PROGRAM MAIN
VAR
	fbEvent:				FB_Event;
	fbEventHandler:			FB_EventHandler;
	fbTcLoggerHandler:		FB_TcLoggerHandler;	
	fbEmergencyHandler:		FB_EmergencyHandler;
	bInit:					BOOL:= TRUE;
	bDebug:					BOOL;
	bInfo:					BOOL;
	bWarning: 				BOOL;
	bError: 				BOOL;
END_VAR

IF bInit THEN
	bInit:= FALSE;
	fbEvent.P_Handler:= fbEventHandler;
	fbEventHandler.P_Next:= fbEmergencyHandler;
	fbEmergencyHandler.P_Next:= fbTcLoggerHandler;
END_IF

fbEvent();
fbEventHandler();
fbTcLoggerHandler();
fbEmergencyHandler();

IF bDebug THEN
	fbEvent.M_Debug('Debug',1);
END_IF

IF bInfo THEN
	fbEvent.M_Info('Warning',2);
END_IF

IF bWarning THEN
	fbEvent.M_Warning('Warning',3);
END_IF

IF bError THEN
	fbEvent.M_Error('Emergency Stop', 4);
END_IF

END_PROGRAM

(* stored: Version 1.1.0.1, ProductVersion 3.1.4024.12
   POU MAIN: Id {e5f7a5a1-3f48-4670-a47b-5f2ccf40d0d9}, SpecialFunc None *)
